FUNCTION_BLOCK ExampleStateMachine IMPLEMENTS I_Init, I_Execute;
VAR
	
	_init: Init(THIS^);

	_ett: EntityStart;
		_ctx: StateContext;
	_ettEnd: EntityEnd;
	
	_post_exe: Execute(THIS^);
END_VAR

PROPERTY Entity : I_Entity
GET
Entity := _ett;
END_GET
END_PROPERTY

(*
If registered, this method will be executed cyclically.
*)
METHOD Execute
VAR_INPUT
	nPhase	: INT;
END_VAR
_ctx.bHmiAcknowledge := FALSE;
END_METHOD

(*
If registered, this method will be executed upon startup.
*)
METHOD Init
VAR_INPUT
	nPhase	: INT;
END_VAR
_ctx.smgr.Request(_ctx.stopped);
END_METHOD

END_FUNCTION_BLOCK

(* stored: Version 1.1.0.1
   POU ExampleStateMachine: Id {b416ac77-f9e5-448c-ae6b-3718da90eacf}, SpecialFunc None
   Property Entity: Id {c30f16a9-26cd-47a8-89ce-c647c5b4d559}
   Get Get: Id {14c13664-5313-4182-b730-759cb62ddf43}
   Method Execute: Id {a304e578-f69c-4edc-aacc-63226b76bdc5}
   Method Init: Id {6ef1b536-d094-4a20-b09d-77b6050a336d} *)
